PROGRAM P_CONTROL
VAR
	bDoors : BOOL;
	State: INT;
	
	
//================	
	// Blink timer
	TIME_ON 			: TIME := T#1S;
	TIME_OFF 			: TIME := T#1S;	
	TIME_FAST_ON 		: TIME := T#250MS;
	TIME_FAST_OFF 		: TIME := T#250MS;
	TIME_SPECIAL_ON 	: TIME := T#50MS;
	TIME_SPECIAL_OFF 	: TIME := T#50MS;	
	
	BlinkTimer_ON: TON;
	BlinkTimer_OFF: TON;
	BlinkTimer_FAST_ON: TON;
	BlinkTimer_FAST_OFF: TON;
	BlinkTimer_SPEC_ON: TON;
	BlinkTimer_SPEC_OFF: TON;
	T_ON : BOOL;
	T_OFF : BOOL := TRUE;	
	T_FAST_ON : BOOL;
	T_FAST_OFF : BOOL := TRUE;	
	T_SPEC_ON : BOOL;
	T_SPEC_OFF : BOOL := TRUE;
//==================

	StateSpecial: INT;
	i: INT;
	Input1_RTRIG: R_TRIG;
	Input2_RTRIG: R_TRIG;
	tempCounter: INT;
	tempCounter2: INT;
	bSwitchToggle: BOOL;
END_VAR


//	A_ButtonBoxes();
//	A_FeedButton();
	Blink();
	Blink_Faster();
	Blink_Special();

ACTION A_Beacons:

END_ACTION

ACTION A_ButtonBoxes:

// Pitäiskö sittenkin olla FBD lajitelma buttonboxien FB?

(*
Input1_RTRIG(CLK:= IN._DI._Label.BTN_Feed);
IF Input1_RTRIG.Q THEN
	A_FeedButton();
END_IF
	
Input2_RTRIG(CLK:= (IN._DI._Label.SWITCH_Left OR IN._DI._Label.SWITCH_Right), Q=> );
IF Input2_RTRIG.Q THEN
	A_Switch();
END_IF

*)
END_ACTION

ACTION Blink:

BlinkTimer_ON(IN:= T_ON , PT:= TIME_ON , Q=> , ET=> );
IF BlinkTimer_ON.Q THEN
	T_ON 	:= GENERAL.BlinkOn:= FALSE;
	T_OFF 	:= TRUE;	
END_IF

BlinkTimer_OFF(IN:= T_OFF , PT:= TIME_OFF , Q=> , ET=> );
IF BlinkTimer_OFF.Q THEN
	T_ON 	:= GENERAL.BlinkOn := TRUE;
	T_OFF	:= FALSE;
END_IF
END_ACTION

ACTION Blink_Faster:


BlinkTimer_FAST_ON(IN:= T_FAST_ON , PT:= TIME_FAST_ON , Q=> , ET=> );
IF BlinkTimer_FAST_ON.Q THEN
	T_FAST_ON	:= GENERAL.BlinkFAST_On:= FALSE;
	T_FAST_OFF 	:= TRUE;	
END_IF

BlinkTimer_FAST_OFF(IN:= T_FAST_OFF , PT:= TIME_FAST_OFF , Q=> , ET=> );
IF BlinkTimer_FAST_OFF.Q THEN
	T_FAST_ON 	:= GENERAL.BlinkFAST_On := TRUE;
	T_FAST_OFF	:= FALSE;
END_IF
END_ACTION

ACTION Blink_Special:

CASE StateSpecial OF
0:

	IF i > 5 THEN
		StateSpecial := 1;
		i := 0;
		ELSE
		BlinkTimer_SPEC_ON(IN:= T_SPEC_ON , PT:= (TIME_SPECIAL_ON*5) , Q=> , ET=> );
		IF BlinkTimer_SPEC_ON.Q THEN
			T_SPEC_ON 	:= GENERAL.BlinkSpecial_ON:= FALSE;
			T_SPEC_OFF 	:= TRUE;	
		END_IF
		
		BlinkTimer_SPEC_OFF(IN:= T_SPEC_OFF , PT:= (TIME_SPECIAL_OFF*5) , Q=> , ET=> );
		IF BlinkTimer_SPEC_OFF.Q THEN
			T_SPEC_ON 	:= GENERAL.BlinkSpecial_ON := TRUE;
			T_SPEC_OFF	:= FALSE;
		i:= i+1;
		END_IF
	END_IF

	1: 

	IF i > 1 THEN
		StateSpecial := 0;
		i := 0;
		ELSE
		BlinkTimer_SPEC_ON(IN:= T_SPEC_ON , PT:= (TIME_SPECIAL_ON*10) , Q=> , ET=> );
		IF BlinkTimer_SPEC_ON.Q THEN
			T_SPEC_ON 	:= GENERAL.BlinkSpecial_ON:= FALSE;
			T_SPEC_OFF 	:= TRUE;	
		END_IF
		
		BlinkTimer_SPEC_OFF(IN:= T_SPEC_OFF , PT:= (TIME_SPECIAL_OFF*10) , Q=> , ET=> );
		IF BlinkTimer_SPEC_OFF.Q THEN
			T_SPEC_ON 	:= GENERAL.BlinkSpecial_ON := TRUE;
			T_SPEC_OFF	:= FALSE;
			i:= i+1;
		END_IF
	END_IF
END_CASE
END_ACTION

END_PROGRAM

(* stored: Version 1.1.0.1, ProductVersion 3.1.4024.10
   POU P_CONTROL: Id {27560784-429a-4cb9-b530-4b903427c533}, SpecialFunc None
   Folder Blinkers: Id {5c25f4da-2386-4bfa-a3e5-3fe24506dcb7}
   Action A_Beacons: Id {9f0f4f38-0331-4251-b759-68adeace686f}
   Action A_ButtonBoxes: Id {78e610f5-06f1-42f9-a722-0082c1dc1f14}
   Action Blink: Id {cf892607-1afc-45ec-8503-4003e9a74f1f}
   Action Blink_Faster: Id {4c379a4c-fd1e-485d-be50-2df9c3314d57}
   Action Blink_Special: Id {ba255915-c92f-459f-ac44-5943878c9a83} *)
